(* 40001 - Read pending logs *)
MODBUS.VARS[8].SlaveAddress:=1;
MODBUS.VARS[8].FunCode:=16#3;
MODBUS.VARS[8].FunAddress:=16#0;
MODBUS.VARS[8].Refresh_Time:=10;
MODBUS.VARS[8].Variable:=ADR(Log_Count);
MODBUS.VARS[8].Variable_Size:=1;
MODBUS.VARS[8].Variable_Mirror:=0;
(* 40011 - Read 1st log entry *)
MODBUS.VARS[9].SlaveAddress:=1;
MODBUS.VARS[9].FunCode:=16#3;
MODBUS.VARS[9].FunAddress:=16#A;
MODBUS.VARS[9].Refresh_Time:=0;
MODBUS.VARS[9].Variable:=ADR(Log_Record);
MODBUS.VARS[9].Variable_Size:=5;
MODBUS.VARS[9].Variable_Mirror:=0;

(****************************************** PDC01 *******)
(* 12028 + 64*ID *)
MODBUS.VARS[10].SlaveAddress:=1;
MODBUS.VARS[10].FunCode:=16#2;
MODBUS.VARS[10].FunAddress:=16#07EB + 64*0;
MODBUS.VARS[10].Refresh_Time:=20;
MODBUS.VARS[10].Variable:=ADR(PDC01.OnOff);
MODBUS.VARS[10].Variable_Size:=1;
MODBUS.VARS[10].Variable_Mirror:=0;
(* 35023 + 250*ID *)
MODBUS.VARS[11].SlaveAddress:=1;
MODBUS.VARS[11].FunCode:=16#4;
MODBUS.VARS[11].FunAddress:=16#139E + 250*0;
MODBUS.VARS[11].Refresh_Time:=20;
MODBUS.VARS[11].Variable:=ADR(PDC01.TSend);
MODBUS.VARS[11].Variable_Size:=1;
MODBUS.VARS[11].Variable_Mirror:=0;
(* 35024 + 250*ID *)
MODBUS.VARS[12].SlaveAddress:=1;
MODBUS.VARS[12].FunCode:=16#4;
MODBUS.VARS[12].FunAddress:=16#139F + 250*0;
MODBUS.VARS[12].Refresh_Time:=20;
MODBUS.VARS[12].Variable:=ADR(PDC01.TRet);
MODBUS.VARS[12].Variable_Size:=1;
MODBUS.VARS[12].Variable_Mirror:=0;
(* 35041 + 250*ID *)
MODBUS.VARS[13].SlaveAddress:=1;
MODBUS.VARS[13].FunCode:=16#4;
MODBUS.VARS[13].FunAddress:=16#13B0 + 250*0;
MODBUS.VARS[13].Refresh_Time:=20;
MODBUS.VARS[13].Variable:=ADR(PDC01.Flow);
MODBUS.VARS[13].Variable_Size:=1;
MODBUS.VARS[13].Variable_Mirror:=0;
(* 35044 + 250*ID *)
MODBUS.VARS[14].SlaveAddress:=1;
MODBUS.VARS[14].FunCode:=16#4;
MODBUS.VARS[14].FunAddress:=16#13B3 + 250*0;
MODBUS.VARS[14].Refresh_Time:=20;
MODBUS.VARS[14].Variable:=ADR(PDC01.Power);
MODBUS.VARS[14].Variable_Size:=1;
MODBUS.VARS[14].Variable_Mirror:=0;
(* 35061 + 250*ID *)
MODBUS.VARS[15].SlaveAddress:=1;
MODBUS.VARS[15].FunCode:=16#4;
MODBUS.VARS[15].FunAddress:=16#13C4 + 250*0;
MODBUS.VARS[15].Refresh_Time:=20;
MODBUS.VARS[15].Variable:=ADR(PDC01.Status);
MODBUS.VARS[15].Variable_Size:=1;
MODBUS.VARS[15].Variable_Mirror:=0;

(****************************************** CAL01 *******)
(* 12028 + 64*ID *)
MODBUS.VARS[16].SlaveAddress:=1;
MODBUS.VARS[16].FunCode:=16#2;
MODBUS.VARS[16].FunAddress:=16#07EB + 64*1;
MODBUS.VARS[16].Refresh_Time:=20;
MODBUS.VARS[16].Variable:=ADR(CAL01.OnOff);
MODBUS.VARS[16].Variable_Size:=1;
MODBUS.VARS[16].Variable_Mirror:=0;
(* 35023 + 250*ID *)
MODBUS.VARS[17].SlaveAddress:=1;
MODBUS.VARS[17].FunCode:=16#4;
MODBUS.VARS[17].FunAddress:=16#139E + 250*1;
MODBUS.VARS[17].Refresh_Time:=20;
MODBUS.VARS[17].Variable:=ADR(CAL01.TSend);
MODBUS.VARS[17].Variable_Size:=1;
MODBUS.VARS[17].Variable_Mirror:=0;
(* 35024 + 250*ID *)
MODBUS.VARS[18].SlaveAddress:=1;
MODBUS.VARS[18].FunCode:=16#4;
MODBUS.VARS[18].FunAddress:=16#139F + 250*1;
MODBUS.VARS[18].Refresh_Time:=20;
MODBUS.VARS[18].Variable:=ADR(CAL01.TRet);
MODBUS.VARS[18].Variable_Size:=1;
MODBUS.VARS[18].Variable_Mirror:=0;
(* 35061 + 250*ID *)
MODBUS.VARS[19].SlaveAddress:=1;
MODBUS.VARS[19].FunCode:=16#4;
MODBUS.VARS[19].FunAddress:=16#13C4 + 250*1;
MODBUS.VARS[19].Refresh_Time:=20;
MODBUS.VARS[19].Variable:=ADR(CAL01.Status);
MODBUS.VARS[19].Variable_Size:=1;
MODBUS.VARS[19].Variable_Mirror:=0;

(****************************************** CAL02*******)
(* 12028 + 64*ID *)
MODBUS.VARS[20].SlaveAddress:=1;
MODBUS.VARS[20].FunCode:=16#2;
MODBUS.VARS[20].FunAddress:=16#07EB + 64*2;
MODBUS.VARS[20].Refresh_Time:=20;
MODBUS.VARS[20].Variable:=ADR(CAL02.OnOff);
MODBUS.VARS[20].Variable_Size:=1;
MODBUS.VARS[20].Variable_Mirror:=0;
(* 35023 + 250*ID *)
MODBUS.VARS[21].SlaveAddress:=1;
MODBUS.VARS[21].FunCode:=16#4;
MODBUS.VARS[21].FunAddress:=16#139E + 250*2;
MODBUS.VARS[21].Refresh_Time:=20;
MODBUS.VARS[21].Variable:=ADR(CAL02.TSend);
MODBUS.VARS[21].Variable_Size:=1;
MODBUS.VARS[21].Variable_Mirror:=0;
(* 35024 + 250*ID *)
MODBUS.VARS[22].SlaveAddress:=1;
MODBUS.VARS[22].FunCode:=16#4;
MODBUS.VARS[22].FunAddress:=16#139F + 250*2;
MODBUS.VARS[22].Refresh_Time:=20;
MODBUS.VARS[22].Variable:=ADR(CAL02.TRet);
MODBUS.VARS[22].Variable_Size:=1;
MODBUS.VARS[22].Variable_Mirror:=0;
(* 35061 + 250*ID *)
MODBUS.VARS[23].SlaveAddress:=1;
MODBUS.VARS[23].FunCode:=16#4;
MODBUS.VARS[23].FunAddress:=16#13C4 + 250*2;
MODBUS.VARS[23].Refresh_Time:=20;
MODBUS.VARS[23].Variable:=ADR(CAL02.Status);
MODBUS.VARS[23].Variable_Size:=1;
MODBUS.VARS[23].Variable_Mirror:=0;

(****************************************** REARM*******)
(* 40244(W) - Reset UnitID *)
MODBUS.VARS[24].SlaveAddress:=1;
MODBUS.VARS[24].FunCode:=16#6;
MODBUS.VARS[24].FunAddress:=16#F3;
MODBUS.VARS[24].Refresh_Time:=0;
MODBUS.VARS[24].Variable:=ADR(Reset_UnitID);
MODBUS.VARS[24].Variable_Size:=1;
MODBUS.VARS[24].Variable_Mirror:=0;
(* 40245(W) - Reset Request *)
MODBUS.VARS[25].SlaveAddress:=1;
MODBUS.VARS[25].FunCode:=16#6;
MODBUS.VARS[25].FunAddress:=16#F4;
MODBUS.VARS[25].Refresh_Time:=0;
MODBUS.VARS[25].Variable:=ADR(Reset_Request);
MODBUS.VARS[25].Variable_Size:=1;
MODBUS.VARS[25].Variable_Mirror:=0;
(* 40246(R) - Status of Reset *)
MODBUS.VARS[26].SlaveAddress:=1;
MODBUS.VARS[26].FunCode:=16#3;
MODBUS.VARS[26].FunAddress:=16#F5;
MODBUS.VARS[26].Refresh_Time:=0;
MODBUS.VARS[26].Variable:=ADR(Reset_Status);
MODBUS.VARS[26].Variable_Size:=1;
MODBUS.VARS[26].Variable_Mirror:=0;


(* Enable variables control *)
MODBUS.VARS_En:=TRUE;
(* End initialization *)
InitOK:=TRUE;
END_ACTION
ACTION Log_Check:
IF Log_Count>0 THEN
	IF Log_Sta=0 THEN
		(* Request log record *)
		MODBUS.VARS[9].Variable_Mirror:=1;
		Log_Sta:=1;
	ELSIF Log_Sta=1 THEN
		(* Check log reading *)
		IF MODBUS.VARS[9].Variable_Mirror=0 THEN
			(* Generate LogEv *)
			Log_Send();
			(* Ack reading *)
			Log_ReadAck:=1;
			MODBUS.VARS[2].Variable_Mirror:=0;
			Log_Sta:=2;
		END_IF
	ELSIF Log_Sta=2 THEN
		(* Check ack writing *)
		IF MODBUS.VARS[2].Variable_Mirror=1 THEN
			(* Update log count *)
			MODBUS.VARS[8].Variable_Mirror:=1;
			Log_Sta:=3;
		END_IF
	ELSIF Log_Sta=3 THEN
		(* Check ack reading *)
		IF MODBUS.VARS[8].Variable_Mirror=0 AND MODBUS.VarProc=FALSE THEN
			Log_Sta:=0;
		END_IF
	END_IF
ELSE
	Log_Sta:=0;
END_IF
END_ACTION
ACTION Log_Send:
(* Generate debug log *)
s1:=RAWTOHEXSTR(pData:=ADR(Log_Record), DataLen:=SIZEOF(Log_Record));
LogEv(EL_Log,EO_GRU,ID,10,s1);

(* Generate decoded event *)
s1:=CONCAT('ID:',WORD_TO_STRING(Log_Record[4]));
i:=Log_Record[2];
IF (i AND 16#0001)<>0 THEN s1:=CONCAT(s1,'-H'); END_IF
IF (i AND 16#0002)<>0 THEN s1:=CONCAT(s1,'-C'); END_IF
IF (i AND 16#0004)<>0 THEN s1:=CONCAT(s1,'-DDC'); END_IF
IF (i AND 16#8000)<>0 THEN s1:=CONCAT(s1,'_Board'); END_IF
IF (i AND 16#0008)<>0 THEN s1:=CONCAT(s1,'_W'); ec:=FALSE;
				      ELSE s1:=CONCAT(s1,'_E'); ec:=TRUE; END_IF
i:=SHR(Log_Record[2] AND 16#7FF0,4);
s1:=CONCAT(s1,WORD_TO_STRING(i));
i:=Log_Record[3] AND 16#3;
IF i=0 OR i=2 THEN
	IF i=0 THEN s1:=CONCAT(s1,'_ON');
		   ELSE s1:=CONCAT(s1,'_EV'); END_IF
	IF ec THEN LogEv(EL_Alarm  ,EO_GRU,ID,13,s1);
		  ELSE LogEv(EL_Wrn,EO_GRU,ID,11,s1); END_IF
ELSIF i=1 THEN
	s1:=CONCAT(s1,'_OFF');
	IF ec THEN LogEv(EL_Log,EO_GRU,ID,14,s1);
		  ELSE LogEv(EL_Log,EO_GRU,ID,12,s1); END_IF
END_IF
END_ACTION
ACTION Reset_Check:
IF Reset_Status=0 THEN
	(* Request status *)
	MODBUS.VARS[26].Variable_Mirror:=1;
ELSE
	(* Check rearm flags *)
	IF PDC01.Rearm THEN
		PDC01.Rearm:=FALSE;
		Reset_UnitID:=0;
		MODBUS.VARS[24].Variable_Mirror:=16#FFFF;
		Reset_Request:=1;
		MODBUS.VARS[25].Variable_Mirror:=16#FFFF;
		Reset_Status:=0;

	ELSIF CAL01.Rearm THEN
		CAL01.Rearm:=FALSE;
		Reset_UnitID:=1;
		MODBUS.VARS[24].Variable_Mirror:=16#FFFF;
		Reset_Request:=1;
		MODBUS.VARS[25].Variable_Mirror:=16#FFFF;
		Reset_Status:=0;

	ELSIF CAL02.Rearm THEN
		CAL02.Rearm:=FALSE;
		Reset_UnitID:=2;
		MODBUS.VARS[24].Variable_Mirror:=16#FFFF;
		Reset_Request:=1;
		MODBUS.VARS[25].Variable_Mirror:=16#FFFF;
		Reset_Status:=0;

	END_IF
END_IF
END_ACTION

(* POU Utils Functions/RAWTOHEXSTR, ST *)
FUNCTION RAWTOHEXSTR : STRING(128)
VAR_INPUT
	pData: POINTER TO BYTE;
	DataLen: BYTE;
END_VAR
VAR
	pt: POINTER TO BYTE;
	xl: BYTE;
END_VAR
pt:=ADR(RAWTOHEXSTR);

xl:=2;

WHILE DataLen>0 AND xl<128 DO

	pt^ := (pData^ / 16#10) + 48 + (((pData^ / 16#10)/10)*7);
	pt:=pt+1;
	pt^ := (pData^ AND 16#0F)  + 48 + (((pData^ AND 16#0F)/10)*7);
	pt:=pt+1;

	xl:=xl+2;

	DataLen:=DataLen-1;
	pData:=pData+1;

END_WHILE

pt^:=0;
END_FUNCTION

(* POU Plant_Objects/obj_PDC_ROBUR_GAHP, ST *)
FUNCTION_BLOCK obj_PDC_ROBUR_GAHP (* POMPA DI CALORE ROBUR GAHP from DDC *)
VAR_INPUT
	(* Settings *)
	ID				: BYTE; (* Index of instanced object *)
	NetID			: WORD; (* Network ID on ROBUR DDC *)

	(* Controls *)
	Rearm			: BOOL; (* 40244=UID(u16-Unit), 40245=1(u16-Reset) *)

	(* States *)
	OnOff			: WORD; (* 12028 + 0*64  *)
	TSend			: INT;	(* 35023 + 0*250 *)
	TRet			: INT;	(* 35024 + 0*250 *)
	Flow			: WORD; (* 35041 + 0*250 = Water flow rate l/h *)
	Power			: WORD; (* 35044 + 0*250 = Power feedback percentage 0-100% *)
	Status			: WORD; (* 35061 + 0*250 = General alarm bits1&0 00:OK 01:LOG 10:WRN 11:ERR *)

END_VAR
VAR_OUTPUT
	(* Visu/Log *)
	Status_Log		: BYTE;
	Status_Vis : DWORD;
END_VAR
VAR
END_VAR
(* Status color *)
   IF (Status AND 16#3)=16#3 THEN Status_Log:=2; Status_Vis:=16#2020F0;
ELSIF (Status AND 16#3)>1    THEN Status_Log:=1; Status_Vis:=16#20F0F0;
              				 ELSE Status_Log:=0; Status_Vis:=SEL(OnOff=1,16#006000,16#20F020);
END_IF
END_FUNCTION_BLOCK

(* POU Plant_Objects/obj_PORT, ST *)
FUNCTION_BLOCK obj_PORT
VAR_INPUT
	(* Settings *)
	ID			: BYTE;
	Peso		 : INT;		(* Peso dell' impulso , serve per avere una lettura immediata dell'unità ingegneristica *)
	TempoTimeOut : TIME;	(* Minuti di inattività per la segnalazione del WRN *)
	PuntoMinX	: INT;  (*Parametri per la scalatura *)
	PuntoMaxX	: INT;
	PuntoMinY	: REAL;
	PuntoMaxY	: REAL;
	Decimali	: BYTE;
	TAP			: INT:=2000;   (* Filtro in msec *)
	INITEV		: BOOL:= TRUE; (* Generate init OK event *)
	SogliaHH	: WORD;    (* Soglia per segnalazione Allarme Extra Range in alto - Solitamente sondo in CC *)
	SogliaHL	: WORD;    (* Soglia per segnalazione Allarme Extra Range in Basso - Solitamente sondo Aperta *)
	SogliaWH	: REAL;    (* Soglia per segnalazione Warning  in alto  *)
	SogliaWL	: REAL;    (* Soglia per segnalazione Warning in basso  *)

	(* Physical inputs *)
	DI_INPUT	: BOOL; (* Ingresso Digitale per il conteggio  *)
	AI_INPUT	: WORD; (* Ingresso Analogico *)
END_VAR
VAR_IN_OUT
    Contatore		: DINT;
    Totalizzatore	: DINT; (* Totale Conteggio x valore peso *)
END_VAR
VAR_OUTPUT
	ValoreScalato	: INT;	(*Valore istantaneo scalato ingresso Analgico *)
	ERR				: BOOL;	(* Segnalazione Errore *)
	WRN				: BOOL;	(* Segnalazione Warning *)

	(* Status *)
	Status_Log	: BYTE;
	Status_Vis 	: DWORD;

END_VAR
VAR
	TRig_DI		: R_TRIG;

	TimeOut		: TON;
	TRigR_TimeOut: R_TRIG;
	TRigL_TimeOut: F_TRIG;

	SegnaleHH: BOOL;
	SegnaleHL: BOOL;
	SegnaleOK: BOOL;

	SegnaleWH: BOOL;
	SegnaleWL: BOOL;

	FiltroWRN:TON;
	FiltroOK:TON;
	FiltroERR:TON;
END_VAR
(**** Gestione ingresso digitale per la contabilizzazzione degli impulsi *****************)

(* TRiggero sul fronte di salita l'ingresso Digitale *)

TRig_DI(CLK:=DI_Input );

(* Conto i fronti di salita  in modo de creare rapporto*)
IF  TRig_DI.Q THEN
	Contatore:=Contatore+1;
	Totalizzatore:=Contatore*Peso;
END_IF


(* Imposto il time out se non c'è movimento sulla linea per il tempo impostato loggo un Warning *)

TimeOut(IN:=NOT DI_Input , PT:=TempoTimeOut, Q=> , ET=> );
TRigR_TimeOut(CLK:= TimeOut.Q  );
TRigL_TimeOut(CLK:= TimeOut.Q  );

		IF  TRigR_TimeOut.Q THEN     (* Condizione di WARNING *)
					WRN:=TRUE;
 					LogEv(EL_Wrn,EO_PORT,ID,5,'Nessun_Movimento'); (********* Morneo ***********)
		END_IF

		IF  TRigL_TimeOut.Q THEN     (* Condizione di Rientro dal WARNING *)
					WRN:=FALSE;
 					LogEv(EL_Log,EO_PORT,ID,1,'');
		END_IF


(**** Gestione ingresso Analogico per la gestione del valore istantaneo  *****************)

(* Verifico che le variabile letta dall'ingresso Analogico  sia dentro i range
ATTENZIONE I LIMITI SPESSO SONO IN WORD VERIFICA  TABELLA MANUALE WAGO  *)

SegnaleHH:=(AI_INPUT>=SogliaHH);
SegnaleHL:=(AI_INPUT<=SogliaHL);
SegnaleOK:=NOT (SegnaleHH OR SegnaleHL);


(* Linerarizzo il segnale di ingresso e la converto in unita ingegneristiche *)
ValoreScalato:=LINEAR(PuntoMinX, PuntoMaxX, AI_INPUT, PuntoMinY, PuntoMaxY,Decimali);

IF SegnaleOK  THEN
	(*  Verifica  e segnalazione Warning *)
	SegnaleWH:=(ValoreScalato>SogliaWH*(EXPT(10, Decimali)));
	SegnaleWL:=(ValoreScalato<SogliaWL*(EXPT(10, Decimali)));

		FiltroWRN(IN:=(SegnaleWH OR SegnaleWL)  , PT:=INT_TO_TIME(TAP) );    (* Filtro su LOG *)
		IF  FiltroWRN.Q THEN     (* Condizione di WARNING *)
			IF NOT WRN THEN
					WRN:=TRUE;
 					LogEv(EL_Wrn,EO_PORT,ID,SEL(ValoreScalato<=SogliaWL,3,2),INT_TO_STRING(ValoreScalato));
			END_IF
		END_IF


	      IF (INITEV OR WRN OR ERR)  AND NOT FiltroWRN.Q THEN

			FiltroWRN(IN:=FALSE  , PT:=INT_TO_TIME(TAP));    (* Resetto il Filtro su LOG WRN  *)
			FiltroERR(IN:=FALSE  , PT:=INT_TO_TIME(TAP));    (* Resetto il Filtro su LOG ERR *)
			INITEV:=FALSE; ERR:=FALSE; WRN:=FALSE;
			LogEv(EL_Log,EO_PORT,ID,1,'');
		END_IF

		 Status_Vis:=16#20F020;    (* Indicazione WEB Visu Sonda OK *)
ELSE
		FiltroERR(IN:=TRUE  , PT:= INT_TO_TIME(TAP) );    (* Filtro su LOG *)
			IF  FiltroERR.Q THEN     (* Condizione di WARNING *)
					IF NOT ERR THEN
						ERR:=TRUE;
						IF SegnaleHH THEN LogEv(EL_Alarm,EO_PORT,ID,6,INT_TO_STRING(ValoreScalato));END_IF;
						IF SegnaleHL THEN LogEv(EL_Alarm,EO_PORT,ID,4,INT_TO_STRING(ValoreScalato));END_IF;
					END_IF
			END_IF

 		Status_Vis:=16#2020F0;   (* Indicazione WEB Visu Sonda KO *)
		Status_Log:=1;

END_IF
END_FUNCTION_BLOCK

(* POU Plant_Objects/obj_TPV, ST *)
FUNCTION_BLOCK obj_TPV
VAR_INPUT
	(* Settings *)
	ID				: BYTE;
	TAP				: BYTE:=4;	   (* Consecutive checks filter *)
	INITEV			: BOOL:= TRUE; (* Generate init OK event *)
	IN_EMIN			: INT :=-2000;
	IN_WMIN			: INT := -500;
	IN_WMAX			: INT :=  500;
	IN_EMAX			: INT := 8500;
	ERR_MIN_SHORT	: BOOL:= TRUE; (* TRUE  ==> EMIN=Short        , EMAX=Disconnected
									  FALSE ==> EMIN=Disconnected , EMAX=Short 		 *)
	(* Physical input *)
	IN				: INT;
END_VAR
VAR_OUTPUT
	WRN:	BOOL;	(* Value in warning range *)
	ERR: 	BOOL; 	(* Value error *)
	HI:		INT;	(* Highest value - cleared by Stat_Reset() action *)
	AVG:	INT; 	(* Average value - updated by Mean() action, cleared by Mean_Reset() action *)
	LOW:	INT;	(* Lowest value  - cleared by Stat_Reset() action *)
END_VAR
VAR
	cnt:	BYTE;
	asum:	DINT;
	acnt:	WORD;
END_VAR
(* Check probe value limits *)
IF IN<=IN_EMIN OR IN>=IN_EMAX THEN
	IF NOT ERR THEN
		cnt:=cnt+1;
		IF cnt>TAP THEN
			cnt:=0;
			ERR:=TRUE; WRN:=FALSE;
			IF ( ERR_MIN_SHORT=TRUE  AND IN<=IN_EMIN ) OR ( ERR_MIN_SHORT=FALSE AND IN>=IN_EMAX ) THEN
				LogEv(EL_Alarm,EO_TPV,ID,5,INT_TO_STRING(IN));
			ELSE
				LogEv(EL_Alarm,EO_TPV,ID,4,INT_TO_STRING(IN));
			END_IF
		END_IF
	END_IF
ELSIF IN<=IN_WMIN OR IN>=IN_WMAX THEN
	IF NOT WRN THEN
		cnt:=cnt+1;
		IF cnt>TAP THEN
			cnt:=0;
			ERR:=FALSE; WRN:=TRUE;
			LogEv(EL_Wrn,EO_TPV,ID,SEL(IN<=IN_WMIN,3,2),INT_TO_STRING(IN));
		END_IF
	END_IF
ELSE
	IF INITEV OR WRN OR ERR THEN
		cnt:=cnt+1;
		IF cnt>TAP THEN
			cnt:=0;
			INITEV:=FALSE; ERR:=FALSE; WRN:=FALSE;
			LogEv(EL_Log,EO_TPV,ID,1,'');
		END_IF
	END_IF
END_IF

(* Average value *)
IF acnt>=60000 THEN
	Mean();
	asum := asum - AVG;
	acnt := acnt - 1;
END_IF

asum := asum + IN;
acnt := acnt + 1;

(* Statistics values *)
IF IN<LOW THEN LOW:=IN; END_IF
IF IN>HI  THEN HI :=IN; END_IF
END_FUNCTION_BLOCK
ACTION Mean:
AVG := DINT_TO_INT(asum/acnt);
END_ACTION
ACTION Mean_Reset:
AVG:=IN;
asum:=IN;
acnt:=1;
END_ACTION
ACTION Stat_Reset:
HI:=IN;
LOW:=IN;
END_ACTION

(* POU Plant_Objects/obj_TPV_SENS, ST *)
FUNCTION_BLOCK obj_TPV_SENS
VAR_INPUT
	(* Settings *)
	ID				: BYTE;
	PuntoMinX		: INT;			(* Parametri per la scalatura *)
	PuntoMaxX		: INT;
	PuntoMinY		: REAL;
	PuntoMaxY		: REAL;
	Decimali		: BYTE;
	SogliaHH		: WORD;			(* Soglia per segnalazione Allarme Extra Range in alto - Solitamente sondo in CC *)
	SogliaHL		: WORD;			(* Soglia per segnalazione Allarme Extra Range in Basso - Solitamente sondo Aperta *)
	SogliaWH		: REAL;			(* Soglia per segnalazione Warning  in alto  *)
	SogliaWL		: REAL;    		(* Soglia per segnalazione Warning in basso  *)
	TAP				: INT:=2000;	(* Filtro in msec *)
	INITEV			: BOOL:= TRUE;	(* Generate init OK event *)

	(* Physical input *)
	AI_INPUT	: WORD;    (* Ingresso Fisico dal modulo Analogico *)

END_VAR
VAR_OUTPUT
	WRN:	BOOL;	(* Segnalazione Warning *)
	ERR: 	BOOL; 	(* Segnalazione Errore *)
	ValoreScalato: INT;
	(* Status *)
	Status_Log	: BYTE;
	Status_Vis 	: DWORD;
END_VAR
VAR

	SegnaleHH: BOOL;
	SegnaleHL: BOOL;
	SegnaleOK: BOOL;

	SegnaleWH: BOOL;
	SegnaleWL: BOOL;

    FiltroWRN:TON;
    FiltroOK:TON;
    FiltroERR:TON;


END_VAR
(* Verifico che le variabile letta dall'ingresso Analogico  sia dentro i range
ATTENZIONE I LIMITI SPESSO SONO IN WORD VERIFICA  TABELLA MANUALE WAGO  *)

SegnaleHH:=(AI_INPUT>=SogliaHH);
SegnaleHL:=(AI_INPUT<=SogliaHL);
SegnaleOK:=NOT (SegnaleHH OR SegnaleHL);

(* Linerarizzo il segnale di ingresso e la converto in unita ingegneristiche *)
ValoreScalato:=LINEAR(PuntoMinX,PuntoMaxX,	AI_INPUT,
					  PuntoMinY,PuntoMaxY,	Decimali);


IF SegnaleOK  THEN

(*  Verifica  e segnalazione Warning *)
	SegnaleWH:=(ValoreScalato>SogliaWH*(EXPT(10, Decimali)));
	SegnaleWL:=(ValoreScalato<SogliaWL*(EXPT(10, Decimali)));

		FiltroWRN(IN:=(SegnaleWH OR SegnaleWL)  , PT:=INT_TO_TIME(TAP) );    (* Filtro su LOG *)
		IF  FiltroWRN.Q THEN     (* Condizione di WARNING *)
			IF NOT WRN THEN
					WRN:=TRUE;
 					LogEv(EL_Wrn,EO_TPV,ID,SEL(ValoreScalato<=SogliaWL,3,2),INT_TO_STRING(ValoreScalato));
			END_IF
		END_IF


	    IF (INITEV OR WRN OR ERR) AND NOT FiltroWRN.Q THEN
			FiltroWRN(IN:=FALSE  , PT:=INT_TO_TIME(TAP));    (* Resetto il Filtro su LOG WRN  *)
			FiltroERR(IN:=FALSE  , PT:=INT_TO_TIME(TAP));    (* Resetto il Filtro su LOG ERR *)
			INITEV:=FALSE; ERR:=FALSE; WRN:=FALSE;
			LogEv(EL_Log,EO_TPV,ID,1,'');
		END_IF

		 Status_Vis:=16#20F020;    (* Indicazione WEB Visu Sonda OK *)
ELSE
		FiltroERR(IN:=TRUE  , PT:= INT_TO_TIME(TAP) );    (* Filtro su LOG *)
			IF  FiltroERR.Q THEN     (* Condizione di WARNING *)
					IF NOT ERR THEN
						ERR:=TRUE;
						IF SegnaleHH THEN LogEv(EL_Alarm,EO_TPV,ID,6,INT_TO_STRING(ValoreScalato));END_IF;
						IF SegnaleHL THEN LogEv(EL_Alarm,EO_TPV,ID,4,INT_TO_STRING(ValoreScalato));END_IF;
					END_IF
			END_IF

 		Status_Vis:=16#2020F0;   (* Indicazione WEB Visu Sonda KO *)

END_IF


(*     Moreno      ********************** Chiedere ad Andrea **

(* Statistics values *)
IF IN<LOW THEN LOW:=IN; END_IF
IF IN>HI  THEN HI :=IN; END_IF
*) 
END_FUNCTION_BLOCK

(* POU PLC_WDT, ST *)
FUNCTION PLC_WDT: DWORD VAR_INPUT dwEvent: DWORD; dwFilter: DWORD; dwOwner: DWORD; END_VAR
LogEv(EL_AlarmStop,EO_SYS,1,10,'Watchdog');
END_FUNCTION

(* POU Utils/RTC_Update, ST *)
FUNCTION RTC_Update : BOOL
VAR
	T: DT;
	TS: STRING;
	TS2: STRING;
	Hour: BYTE;
	Minute: BYTE;
END_VAR
(* Get RTC time *)
T:=SysRtcGetTime(TRUE);
Sys.Time_CT_DT:=T;
(* Calculate variables *)
TS:=DT_TO_STRING(T);
Sys.Time_LogString:=DELETE(STR:=TS, LEN:=3, POS:=1);
TS2:=MID(STR:=TS, LEN:=4, POS:= 4); Sys.Time_Year 	:=STRING_TO_WORD(TS2);
TS2:=MID(STR:=TS, LEN:=2, POS:= 9); Sys.Time_Month	:=STRING_TO_BYTE(TS2);
TS2:=MID(STR:=TS, LEN:=2, POS:=12); Sys.Time_Day  	:=STRING_TO_BYTE(TS2);
Sys.Time_CT_Day:=(32*(Sys.Time_Month-1)+Sys.Time_Day-1);
TS2:=MID(STR:=TS, LEN:=2, POS:=15); Hour			:=STRING_TO_BYTE(TS2);
TS2:=MID(STR:=TS, LEN:=2, POS:=18); Minute		 	:=STRING_TO_BYTE(TS2);
Sys.Time_CT_Quarter:=Hour*4+(Minute/15);
END_FUNCTION

(* POU Utils Functions/TONOF, ST *)
FUNCTION_BLOCK TONOF
VAR_INPUT
	IN		: BOOL;
	PT_ON	: TIME; (* time to pass, before OUT is set *)
	PT_OF	: TIME; (* time to pass, before OUT is reset *)
END_VAR
VAR_OUTPUT
	OUT		: BOOL;
END_VAR
VAR
	timer	: TON;
END_VAR
IF IN<>OUT THEN
	timer(IN:=TRUE,PT:=SEL(IN,PT_OF,PT_ON));
	IF timer.Q THEN OUT:=IN; END_IF
ELSE
	timer(IN:=FALSE);
END_IF
END_FUNCTION_BLOCK

(* Visualisation PLC_VISU
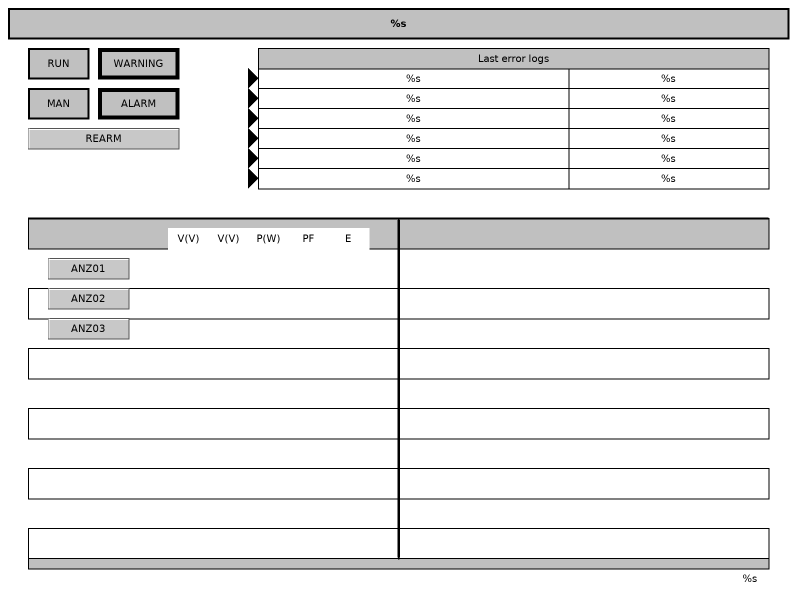
rectangle at (10,10)-(791,41): text "%s"; shows .Plant_NAME
rectangle at (520,570)-(761,591): text "%s"; shows Sys.Time_LogString
rounded rectangle at (30,50)-(91,81): text "RUN"; alarm colour if NOT Mode_Manual; runs INTERN ASSIGN Mode_Manual:=(FALSE)
rounded rectangle at (30,90)-(91,121): text "MAN"; alarm colour if Mode_Manual; runs INTERN ASSIGN Mode_Manual:=(TRUE)
rectangle at (570,70)-(771,91): text "%s"; shows Sys.LastLogs_Msg[0]
polygon at (250,170)-(260,190): invisible if Sys.LastLogs_Idx<>0
rectangle at (570,90)-(771,111): text "%s"; shows Sys.LastLogs_Msg[1]
polygon at (250,70)-(260,90): invisible if Sys.LastLogs_Idx<>1
rectangle at (570,110)-(771,131): text "%s"; shows Sys.LastLogs_Msg[2]
polygon at (250,90)-(260,110): invisible if Sys.LastLogs_Idx<>2
rectangle at (570,130)-(771,151): text "%s"; shows Sys.LastLogs_Msg[3]
polygon at (250,110)-(260,130): invisible if Sys.LastLogs_Idx<>3
rectangle at (570,150)-(771,171): text "%s"; shows Sys.LastLogs_Msg[4]
polygon at (250,130)-(260,150): invisible if Sys.LastLogs_Idx<>4
rectangle at (570,170)-(771,191): text "%s"; shows Sys.LastLogs_Msg[5]
polygon at (250,150)-(260,170): invisible if Sys.LastLogs_Idx<>5
rectangle at (260,70)-(571,91): text "%s"; shows Sys.LastLogs_Dat[0]
rectangle at (260,90)-(571,111): text "%s"; shows Sys.LastLogs_Dat[1]
rectangle at (260,110)-(571,131): text "%s"; shows Sys.LastLogs_Dat[2]
rectangle at (260,130)-(571,151): text "%s"; shows Sys.LastLogs_Dat[3]
rectangle at (260,150)-(571,171): text "%s"; shows Sys.LastLogs_Dat[4]
rectangle at (260,170)-(571,191): text "%s"; shows Sys.LastLogs_Dat[5]
rectangle at (100,90)-(181,121): text "ALARM"; alarm colour if Sys.Alarm; runs INTERN ASSIGN Mode_Manual:=(FALSE)
rectangle at (100,50)-(181,81): text "WARNING"; alarm colour if Sys.Warning; runs INTERN ASSIGN Mode_Manual:=(TRUE)
button at (30,130)-(181,151): text "REARM"; runs INTERN ASSIGN Sys.Alarm:=(FALSE);INTERN ASSIGN Sys.Warning:=(FALSE)
button at (50,260)-(131,281): text "ANZ01"
rectangle at (260,50)-(771,71): text "Last error logs"
button at (50,290)-(131,311): text "ANZ02"
rectangle at (170,230)-(211,251): text "V(V)"
rectangle at (250,230)-(291,251): text "P(W)"
rectangle at (290,230)-(331,251): text "PF"
rectangle at (330,230)-(371,251): text "E"
rectangle at (210,230)-(251,251): text "V(V)"
button at (50,320)-(131,341): text "ANZ03"
9 more shapes without text or variables
5 elements of other kinds (tables, trends, ...) not read
*)
